// TIA Portal project "ProcessVisualization.TankSimulation" (V14)

(* hardware
DEVICE "S7-1200 station_2"  S7-1200 Station
   slot 0: "Rack_0"  S7-1200 Rack  Rack  V1.0
   slot 1: "TankSimulation"  CPU 1212C DC/DC/Rly  6ES7 212-1HE31-0XB0  V3.0
*)

// ===== PLC "TankSimulation"  CPU 1212C DC/DC/Rly =====

DATA_BLOCK "Parameters"   // DB1
{ S7_Optimized_Access := 'FALSE' }
VERSION : 0.1
   VAR
      StartPump : Bool;
      StopPump : Bool;
      PumpRunning : Bool;
      HighLevelLimitSwitch : Bool;
      LowLevelLimitSwitch : Bool;
      TankLevel : Int;
      StartAuto : Bool;
      AutoRunning : Bool;
      StopAuto : Bool;
      FlowSpeed : Int := 1;
      PumpSpeed : Int := 2;
   END_VAR
BEGIN
END_DATA_BLOCK

DATA_BLOCK "TankSimulationDb"   // DB2
{ S7_Optimized_Access := 'TRUE' }
VERSION : 0.1
// stored: InstanceOfName TankSimulation
"TankSimulation"
BEGIN
END_DATA_BLOCK

FUNCTION_BLOCK "TankSimulation"   // FB1, LAD
{ S7_Optimized_Access := 'TRUE' }
VERSION : 0.1
   VAR
      Clock100ms : Bool;
      "Timer" : IEC_TIMER;
   END_VAR
BEGIN

REGION Network 1: Clock 100ms
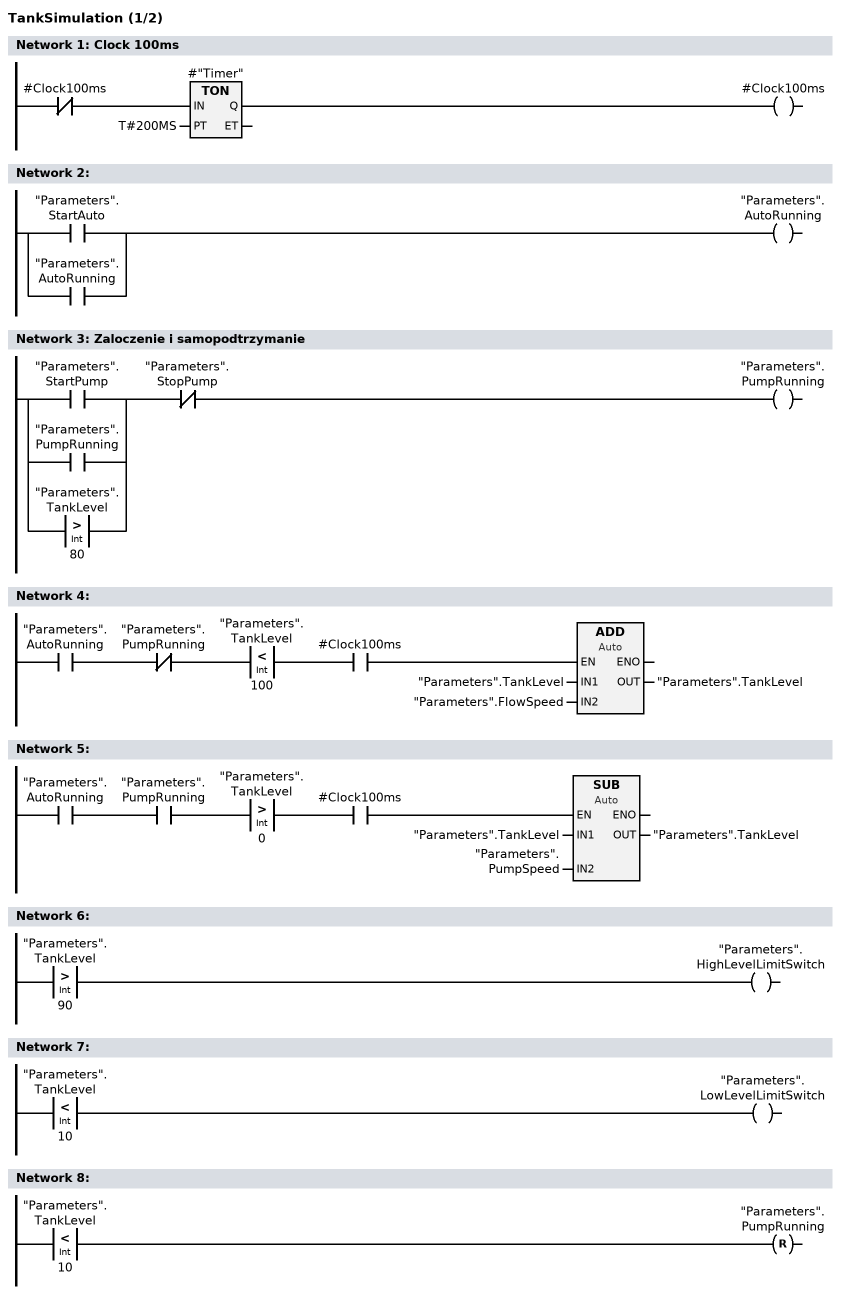
   #"Timer".TON(IN := NOT #Clock100ms, PT := T#200MS);
   #Clock100ms := #"Timer".Q;
END_REGION

REGION Network 2
   RUNG wire#powerrail
      Contact( "Parameters".StartAuto )
      wire#w1
      Coil( "Parameters".AutoRunning )
   END_RUNG
   RUNG wire#powerrail
      Contact( "Parameters".AutoRunning )
   END_RUNG wire#w1
   // the same network as SCL:
   "Parameters".AutoRunning := "Parameters".StartAuto OR "Parameters".AutoRunning;
END_REGION

REGION Network 3: Zaloczenie i samopodtrzymanie
   RUNG wire#powerrail
      Contact( "Parameters".StartPump )
      wire#w1
      I_Contact( "Parameters".StopPump )
      Coil( "Parameters".PumpRunning )
   END_RUNG
   RUNG wire#powerrail
      Contact( "Parameters".PumpRunning )
   END_RUNG wire#w1
   RUNG wire#powerrail
      { S7_Templates := "SrcType := Int" } GT_Contact(in1 := "Parameters".TankLevel, in2 := 80)
   END_RUNG wire#w1
   // the same network as SCL:
   "Parameters".PumpRunning := ("Parameters".StartPump OR "Parameters".PumpRunning OR ("Parameters".TankLevel > 80)) AND NOT "Parameters".StopPump;
END_REGION

REGION Network 4
   RUNG wire#powerrail
      Contact( "Parameters".AutoRunning )
      I_Contact( "Parameters".PumpRunning )
      { S7_Templates := "SrcType := Int" } LT_Contact(in1 := "Parameters".TankLevel, in2 := 100)
      Contact( #Clock100ms )
      { S7_GenerateENO := "TRUE" } Add(in1 := "Parameters".TankLevel, in2 := "Parameters".FlowSpeed, out => "Parameters".TankLevel)
   END_RUNG
   // the same network as SCL:
   IF "Parameters".AutoRunning AND NOT "Parameters".PumpRunning AND ("Parameters".TankLevel < 100) AND #Clock100ms THEN
       "Parameters".TankLevel := "Parameters".TankLevel + "Parameters".FlowSpeed;
   END_IF;
END_REGION

REGION Network 5
   RUNG wire#powerrail
      Contact( "Parameters".AutoRunning )
      Contact( "Parameters".PumpRunning )
      { S7_Templates := "SrcType := Int" } GT_Contact(in1 := "Parameters".TankLevel, in2 := 0)
      Contact( #Clock100ms )
      { S7_GenerateENO := "TRUE" } Sub(in1 := "Parameters".TankLevel, in2 := "Parameters".PumpSpeed, out => "Parameters".TankLevel)
   END_RUNG
   // the same network as SCL:
   IF "Parameters".AutoRunning AND "Parameters".PumpRunning AND ("Parameters".TankLevel > 0) AND #Clock100ms THEN
       "Parameters".TankLevel := "Parameters".TankLevel - "Parameters".PumpSpeed;
   END_IF;
END_REGION

REGION Network 6
   RUNG wire#powerrail
      { S7_Templates := "SrcType := Int" } GT_Contact(in1 := "Parameters".TankLevel, in2 := 90)
      Coil( "Parameters".HighLevelLimitSwitch )
   END_RUNG
   // the same network as SCL:
   "Parameters".HighLevelLimitSwitch := "Parameters".TankLevel > 90;
END_REGION

REGION Network 7
   RUNG wire#powerrail
      { S7_Templates := "SrcType := Int" } LT_Contact(in1 := "Parameters".TankLevel, in2 := 10)
      Coil( "Parameters".LowLevelLimitSwitch )
   END_RUNG
   // the same network as SCL:
   "Parameters".LowLevelLimitSwitch := "Parameters".TankLevel < 10;
END_REGION

REGION Network 8
   RUNG wire#powerrail
      { S7_Templates := "SrcType := Int" } LT_Contact(in1 := "Parameters".TankLevel, in2 := 10)
      R_Coil( "Parameters".PumpRunning )
   END_RUNG
   // the same network as SCL:
   IF "Parameters".TankLevel < 10 THEN "Parameters".PumpRunning := FALSE; END_IF;
END_REGION

REGION Network 9
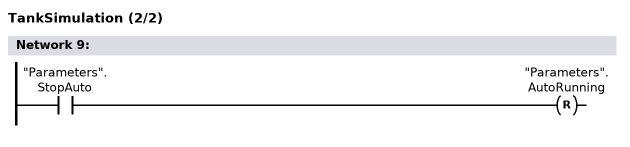
   RUNG wire#powerrail
      Contact( "Parameters".StopAuto )
      R_Coil( "Parameters".AutoRunning )
   END_RUNG
   // the same network as SCL:
   IF "Parameters".StopAuto THEN "Parameters".AutoRunning := FALSE; END_IF;
END_REGION
END_FUNCTION_BLOCK

ORGANIZATION_BLOCK "Main"   // OB1, LAD, ProgramCycle
TITLE = "Main Program Sweep (Cycle)"
{ S7_Optimized_Access := 'TRUE' }
VERSION : 0.1
   VAR_INPUT
      Initial_Call : Bool;   // Initial call of this OB
      Remanence : Bool;   // =True, if remanent data are available
   END_VAR
BEGIN

REGION Network 1
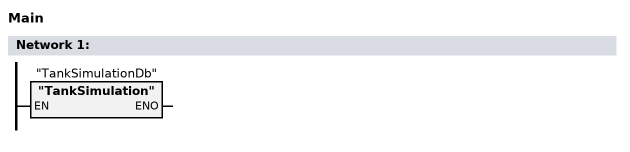
   RUNG wire#powerrail
      "TankSimulationDb"()
   END_RUNG
   // the same network as SCL:
   "TankSimulationDb"();   // "TankSimulation"
END_REGION
END_ORGANIZATION_BLOCK